Staubli VAL3: CirClePoint.pgx

public program CirClePoint(trsf x_trCenter, num x_nDia, trsf& x_trDest[], bool& x_bRes)
  local num l_nNum
  local frame l_fFrame
  local point l_pP
begin
  //由圆心直径获得圆的四个点
  //是通过逆时针来获得

  x_bRes=false

  if x_nDia<=0
    return
  endIf

  link(l_fFrame,world)
  l_fFrame.trsf=x_trCenter
  link(l_pP,l_fFrame)


  //第一个点
  l_pP.trsf={0,0,0,0,0,0}
  l_pP.trsf.y=-x_nDia/2
  x_trDest[0]=position(l_pP,world)


  //第二个点
  l_pP.trsf={0,0,0,0,0,0}
  l_pP.trsf.x=x_nDia/2
  x_trDest[1]=position(l_pP,world)



  //第三个点
  l_pP.trsf={0,0,0,0,0,0}
  l_pP.trsf.y=x_nDia/2
  x_trDest[2]=position(l_pP,world)


  //第四个点
  l_pP.trsf={0,0,0,0,0,0}
  l_pP.trsf.x=-x_nDia/2
  x_trDest[3]=position(l_pP,world)

   x_trDest[4]= x_trDest[0]





  //圆心点
  x_trDest[20]=x_trCenter

  x_bRes=true

  //辅助点
  l_pP.trsf={0,0,0,0,0,0}
  l_pP.trsf.y=-x_nDia/2
    l_pP.trsf.x=x_nDia/2
  x_trDest[9]=position(l_pP,world)






end
